FUNCTION_BLOCK Bomba_Higienizacao_HMI (* Service Interface Function Block Type *)
  (* Standard: 61499-2 *)
  (* Version 0.0, 04/03/2026, template *)
  PACKAGE Hidryco.HidrycoLib;
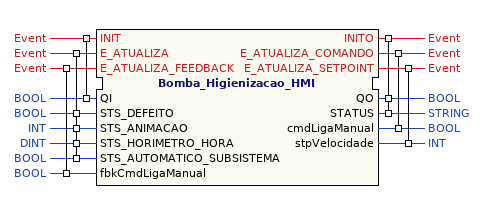
  EVENT_INPUT
    INIT WITH QI;
    E_ATUALIZA WITH STS_DEFEITO, STS_ANIMACAO, STS_HORIMETRO_HORA, STS_AUTOMATICO_SUBSISTEMA;
    E_ATUALIZA_FEEDBACK WITH fbkCmdLigaManual;
  END_EVENT
  EVENT_OUTPUT
    INITO WITH QO, STATUS;
    E_ATUALIZA_COMANDO WITH cmdLigaManual;
    E_ATUALIZA_SETPOINT WITH stpVelocidade;
  END_EVENT
  VAR_INPUT
    QI : BOOL;
    STS_DEFEITO : BOOL;
    STS_ANIMACAO : INT;
    STS_HORIMETRO_HORA : DINT;
    STS_AUTOMATICO_SUBSISTEMA : BOOL;
    fbkCmdLigaManual : BOOL;
  END_VAR
  VAR_OUTPUT
    QO : BOOL; (* Event Output Qualifier *)
    STATUS : STRING; (* Service Status *)
    cmdLigaManual : BOOL;
    stpVelocidade : INT;
  END_VAR
  SERVICE /
    SEQUENCE 
    END_SEQUENCE
  END_SERVICE
END_FUNCTION_BLOCK
